// TIA Portal V20 export
VAR_GLOBAL   // PLC tag table "SS2"
   SS2_Column_Buzzer AT %Q2203.7 : Bool;
   SS2_Column_Red AT %Q2203.6 : Bool;
   SS2_Column_Yellow AT %Q2203.5 : Bool;
   SS2_Column_Green AT %Q2203.4 : Bool;
   ST23_Hydraulic_Rollers_Down AT %Q2200.0 : Bool;
   ST23_Hydraulic_Rollers_Up AT %Q2200.1 : Bool;
   ST23_Modules_Up AT %Q2200.2 : Bool;
   reserve AT %Q2200.3 : Bool;
   "reserve(1)" AT %Q2200.4 : Bool;
   ST24_Hydraulic_Rollers_Down AT %Q2200.5 : Bool;
   ST24_Hydraulic_Rollers_Up AT %Q2200.6 : Bool;
   ST24_Modules_Up AT %Q2200.7 : Bool;
   "reserve(2)" AT %Q2201.0 : Bool;
   "reserve(3)" AT %Q2201.1 : Bool;
   ST25_Hydraulic_Rollers_Down AT %Q2201.2 : Bool;
   ST25_Hydraulic_Rollers_Up AT %Q2201.3 : Bool;
   ST25_Modules_Up AT %Q2201.4 : Bool;
   "reserve(4)" AT %Q2201.5 : Bool;
   "reserve(5)" AT %Q2201.6 : Bool;
   ST23_MOD1_Sen11 AT %I2200.0 : Bool;
   ST23_MOD1_Sen12 AT %I2200.1 : Bool;
   ST23_MOD1_Sen21 AT %I2200.2 : Bool;
   ST23_MOD1_Sen22 AT %I2200.3 : Bool;
   ST23_MOD2_Sen11 AT %I2200.4 : Bool;
   ST23_MOD2_Sen12 AT %I2200.5 : Bool;
   ST23_MOD2_Sen21 AT %I2200.6 : Bool;
   ST23_MOD2_Sen22 AT %I2200.7 : Bool;
   ST23_MOD3_Sen11 AT %I2201.0 : Bool;
   ST23_MOD3_Sen12 AT %I2201.1 : Bool;
   ST23_MOD3_Sen21 AT %I2201.2 : Bool;
   ST23_MOD3_Sen22 AT %I2201.3 : Bool;
   ST23_PAL_Sen11 AT %I2201.4 : Bool;
   ST23_PAL_Sen12 AT %I2201.5 : Bool;
   ST23_PAL_Sen21 AT %I2201.6 : Bool;
   ST23_PAL_Sen22 AT %I2201.7 : Bool;
   ST24_MOD1_Sen11 AT %I2202.0 : Bool;
   ST24_MOD1_Sen12 AT %I2202.1 : Bool;
   ST24_MOD1_Sen21 AT %I2202.2 : Bool;
   ST24_MOD1_Sen22 AT %I2202.3 : Bool;
   ST24_MOD2_Sen11 AT %I2202.4 : Bool;
   ST24_MOD2_Sen12 AT %I2202.5 : Bool;
   ST24_MOD2_Sen21 AT %I2202.6 : Bool;
   ST24_MOD2_Sen22 AT %I2202.7 : Bool;
   ST24_MOD3_Sen11 AT %I2203.0 : Bool;
   ST24_MOD3_Sen12 AT %I2203.1 : Bool;
   ST24_MOD3_Sen21 AT %I2203.2 : Bool;
   ST24_MOD3_Sen22 AT %I2203.3 : Bool;
   ST24_PAL_Sen11 AT %I2203.4 : Bool;
   ST24_PAL_Sen12 AT %I2203.5 : Bool;
   ST24_PAL_Sen21 AT %I2203.6 : Bool;
   ST24_PAL_Sen22 AT %I2203.7 : Bool;
   ST23_Drivers_Rollers_Up AT %Q2202.0 : Bool;
   ST24_Drivers_Rollers_Up AT %Q2202.1 : Bool;
   ST25_Drivers_Rollers_Up AT %Q2202.2 : Bool;
   ST25_MOD1_Sen11 AT %I2204.0 : Bool;
   ST25_MOD1_Sen12 AT %I2204.1 : Bool;
   ST25_MOD1_Sen21 AT %I2204.2 : Bool;
   ST25_MOD1_Sen22 AT %I2204.3 : Bool;
   ST25_MOD2_Sen11 AT %I2204.4 : Bool;
   ST25_MOD2_Sen12 AT %I2204.5 : Bool;
   ST25_MOD2_Sen21 AT %I2204.6 : Bool;
   ST25_MOD2_Sen22 AT %I2204.7 : Bool;
   ST25_MOD3_Sen11 AT %I2205.0 : Bool;
   ST25_MOD3_Sen12 AT %I2205.1 : Bool;
   ST25_MOD3_Sen21 AT %I2205.2 : Bool;
   ST25_MOD3_Sen22 AT %I2205.3 : Bool;
   ST25_PAL_Sen11 AT %I2205.4 : Bool;
   ST25_PAL_Sen12 AT %I2205.5 : Bool;
   ST25_PAL_Sen21 AT %I2205.6 : Bool;
   ST25_PAL_Sen22 AT %I2205.7 : Bool;
   ST23_25_Y0 AT %Q2250.0 : Bool;
   Estop_SS2_ChA AT %I2255.0 : Bool;
   Estop_SS2_ChB AT %I2255.4 : Bool;
   ST23_DR_a_Up AT %I2206.0 : Bool;
   ST23_DR_a_Down AT %I2206.1 : Bool;
   ST23_DR_b_Up AT %I2206.2 : Bool;
   ST23_DR_b_Down AT %I2206.3 : Bool;
   ST24_DR_a_Up AT %I2206.4 : Bool;
   ST24_DR_a_Down AT %I2206.5 : Bool;
   ST24_DR_b_Up AT %I2206.6 : Bool;
   ST24_DR_b_Down AT %I2206.7 : Bool;
   ST25_DR_a_Up AT %I2207.0 : Bool;
   ST25_DR_a_Down AT %I2207.1 : Bool;
   ST25_DR_b_Up AT %I2207.2 : Bool;
   ST25_DR_b_Down AT %I2207.3 : Bool;
   ST23_MOD1_Wib_Contactor AT %Q2202.3 : Bool;
   ST25_MOD1_Wib_Contactor AT %Q2202.4 : Bool;
   ST24_MOD1_Wib_Contactor AT %Q2202.5 : Bool;
   ST23_MOD2_Wib_Contactor AT %Q2202.6 : Bool;
   ST25_MOD2_Wib_Contactor AT %Q2202.7 : Bool;
   ST24_MOD2_Wib_Contactor AT %Q2203.0 : Bool;
   ST23_MOD3_Wib_Contactor AT %Q2203.1 : Bool;
   ST25_MOD3_Wib_Contactor AT %Q2203.2 : Bool;
   ST24_MOD3_Wib_Contactor AT %Q2203.3 : Bool;
END_VAR
